FUNCTION_BLOCK FutureMCResetCreator IMPLEMENTS InterfaceTaskCreator
VAR_INPUT
END_VAR
VAR_OUTPUT
END_VAR
VAR
	_axis: REFERENCE TO AXIS_REF;
END_VAR

{warning 'add method implementation '}
METHOD create_future : InterfaceFuture
VAR_INPUT
	(* Specify future name*)
	future_name	: STRING;
END_VAR
VAR
	_p_future : POINTER TO FutureMCReset;
END_VAR
_p_future := __NEW(FutureMCReset);
_p_future^.future_name := future_name;
_p_future^.set_parameters(_axis);
create_future := _p_future^;
END_METHOD

{warning 'add method implementation '}
METHOD destroy_future : InterfaceFuture
VAR_INPUT
	(* Specify future instance whtat you want to delete.*)
	future	: InterfaceFuture;
END_VAR
VAR
	_p_future : POINTER TO FutureMCReset;
END_VAR
IF __QUERYPOINTER(future, _p_future) THEN
	__DELETE(_p_future);
	IF _p_future = 0  THEN
		destroy_future := 0;
	END_IF
END_IF
END_METHOD

METHOD set_parameters : BOOL
VAR_INPUT
	axis : REFERENCE TO AXIS_REF;
END_VAR
_axis REF= axis;
END_METHOD

END_FUNCTION_BLOCK

(* stored: Version 1.1.0.1, ProductVersion 3.1.4024.15
   POU FutureMCResetCreator: Id {4b617ec0-6e38-4018-982f-d56eab5d2352}, SpecialFunc None
   Method create_future: Id {6b65e0b4-f650-4e62-96fb-3435a29969c8}
   Method destroy_future: Id {9546b0b8-387a-4e24-85b8-a19563cf1a23}
   Method set_parameters: Id {9ad52aad-61d1-4f99-8aaf-d2c89cd99e29} *)
